(* IEC 61131-3 sources: Palletizer_Control_with_Automation_Studio/Palletizer/Logical/Libraries/Filter, 3 files *)

(* ---- filter_FB.st ---- *)
(* TODO: Add your comment here *)
FUNCTION_BLOCK filter_FB

	IF (OperationType = INIT) THEN
		Delay := 0;
	END_IF;

	IF (Clock AND (Delay > 0)) THEN
		Delay := Delay - 1;
	END_IF;

	IF  (Delay = 0) THEN
		DelayedSignal := Signal;
	END_IF;

	IF  (Signal = DelayedSignal) THEN
		IF  (Signal) THEN
			Delay := DeactivationDelay;
		ELSE
			Delay := ActivationDelay;
		END_IF;
	END_IF

END_FUNCTION_BLOCK

(* ---- Constants.var ---- *)
VAR CONSTANT

END_VAR

(* ---- Filter.fun ---- *)
{REDUND_ERROR} {REDUND_UNREPLICABLE} FUNCTION_BLOCK filter_FB (*TODO: Add your comment here*) (*$GROUP=User,$CAT=User,$GROUPICON=User.png,$CATICON=User.png*)
	VAR_INPUT
		OperationType : {REDUND_UNREPLICABLE} INT;
		Clock : {REDUND_UNREPLICABLE} BOOL;
		Signal : {REDUND_UNREPLICABLE} BOOL;
		DeactivationDelay : {REDUND_UNREPLICABLE} INT;
		ActivationDelay : {REDUND_UNREPLICABLE} INT;
	END_VAR
	VAR_OUTPUT
		DelayedSignal : {REDUND_UNREPLICABLE} BOOL;
	END_VAR
	VAR
		Delay : {REDUND_UNREPLICABLE} INT;
	END_VAR
END_FUNCTION_BLOCK
